FUNCTION_BLOCK Lift (* Composite Function Block Type *)
  (* Standard: 61499-2 *)
  (* Version 0.0, 6/3/2016, Andrei, nxtControl GmbH, template *)
  PACKAGE Main;
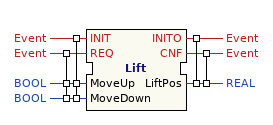
  EVENT_INPUT
    INIT WITH MoveUp, MoveDown; (* Initialization Request *)
    REQ WITH MoveUp, MoveDown; (* Normal Execution Request *)
  END_EVENT
  EVENT_OUTPUT
    INITO WITH LiftPos; (* Initialization Confirm *)
    CNF WITH LiftPos; (* Execution Confirmation *)
  END_EVENT
  VAR_INPUT
    MoveUp : BOOL; (* Input event qualifier *)
    MoveDown : BOOL;
  END_VAR
  VAR_OUTPUT
    LiftPos : REAL; (* Output event qualifier *)
  END_VAR
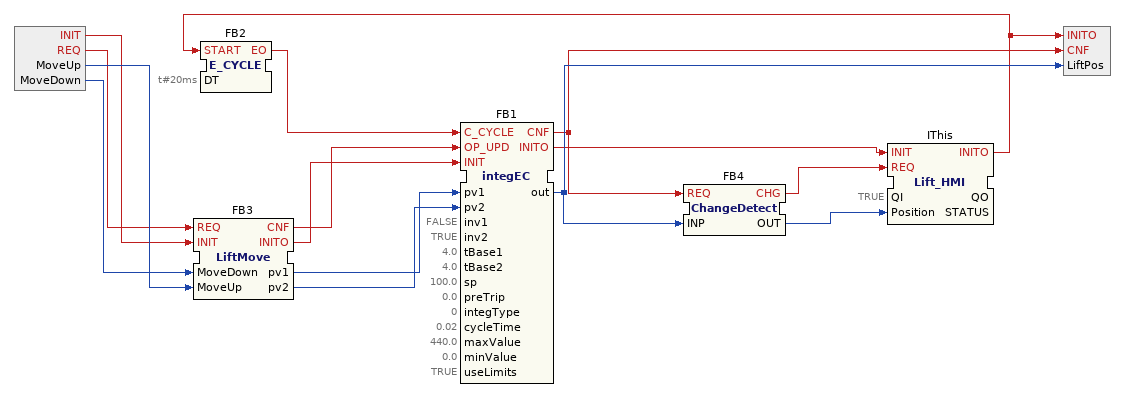
  FBS
    FB2 : E_CYCLE(DT := t#20ms);
    FB4 : ChangeDetect;
    IThis : Lift_HMI(QI := TRUE);
    FB3 : LiftMove;
    FB1 : integEC(inv1 := FALSE, inv2 := TRUE, tBase1 := 4.0, tBase2 := 4.0, sp := 100.0, preTrip := 0.0, integType := 0, cycleTime := 0.02, maxValue := 440.0, minValue := 0.0, useLimits := TRUE);
  END_FBS
  EVENT_CONNECTIONS
    FB2.EO TO FB1.C_CYCLE;
    REQ TO FB3.REQ;
    FB3.CNF TO FB1.OP_UPD;
    INIT TO FB3.INIT;
    FB3.INITO TO FB1.INIT;
    FB1.CNF TO FB4.REQ;
    FB1.INITO TO IThis.INIT;
    FB4.CHG TO IThis.REQ;
    IThis.INITO TO INITO;
    IThis.INITO TO FB2.START;
    FB1.CNF TO CNF;
  END_CONNECTIONS
  DATA_CONNECTIONS
    FB3.pv1 TO FB1.pv1;
    FB3.pv2 TO FB1.pv2;
    MoveDown TO FB3.MoveDown;
    MoveUp TO FB3.MoveUp;
    FB1.out TO FB4.INP;
    FB4.OUT TO IThis.Position;
    FB1.out TO LiftPos;
  END_CONNECTIONS
END_FUNCTION_BLOCK
